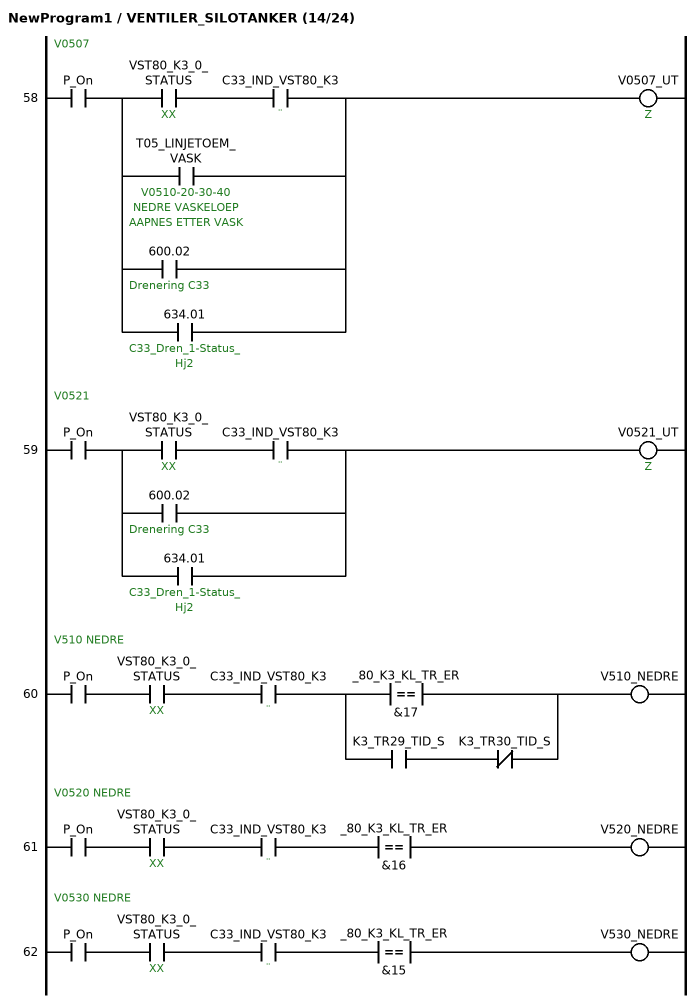
; [picture p864: NewProgram1 / VENTILER_SILOTANKER, rungs 58-62]
; rung 58: V0507
LD P_On
LD VST80_K3_0_STATUS  ; XX
AND C33_IND_VST80_K3  ; ¨
OR T05_LINJETOEM_VASK  ; V0510-20-30-40 NEDRE VASKELOEP AAPNES ETTER VASK
OR 600.02  ; Drenering C33
OR 634.01  ; C33_Dren_1-Status_Hj2
ANDLD
OUT V0507_UT  ; Z
; rung 59: V0521
LD P_On
LD VST80_K3_0_STATUS  ; XX
AND C33_IND_VST80_K3  ; ¨
OR 600.02  ; Drenering C33
OR 634.01  ; C33_Dren_1-Status_Hj2
ANDLD
OUT V0521_UT  ; Z
; rung 60: V510 NEDRE
LD P_On
AND VST80_K3_0_STATUS  ; XX
AND C33_IND_VST80_K3  ; ¨
LD=(300) _80_K3_KL_TR_ER &17
LD K3_TR29_TID_S
ANDNOT K3_TR30_TID_S
ORLD
ANDLD
OUT V510_NEDRE
; rung 61: V0520 NEDRE
LD P_On
AND VST80_K3_0_STATUS  ; XX
AND C33_IND_VST80_K3  ; ¨
AND=(300) _80_K3_KL_TR_ER &16
OUT V520_NEDRE
; rung 62: V0530 NEDRE
LD P_On
AND VST80_K3_0_STATUS  ; XX
AND C33_IND_VST80_K3  ; ¨
AND=(300) _80_K3_KL_TR_ER &15
OUT V530_NEDRE

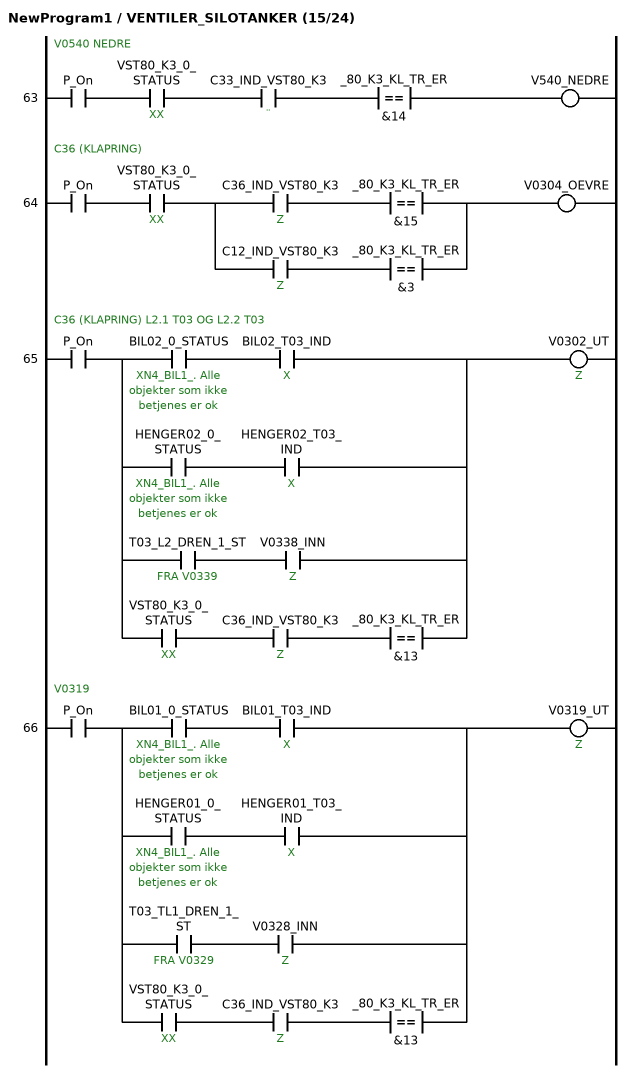
; rung 63: V0540 NEDRE
LD P_On
AND VST80_K3_0_STATUS  ; XX
AND C33_IND_VST80_K3  ; ¨
AND=(300) _80_K3_KL_TR_ER &14
OUT V540_NEDRE
; rung 64: C36 (KLAPRING)
LD P_On
AND VST80_K3_0_STATUS  ; XX
LD C36_IND_VST80_K3  ; Z
AND=(300) _80_K3_KL_TR_ER &15
LD C12_IND_VST80_K3  ; Z
AND=(300) _80_K3_KL_TR_ER &3
ORLD
ANDLD
OUT V0304_OEVRE
; rung 65: C36 (KLAPRING) L2.1 T03 OG L2.2 T03
LD P_On
LD BIL02_0_STATUS  ; XN4_BIL1_. Alle objekter som ikke betjenes er ok
AND BIL02_T03_IND  ; X
LD HENGER02_0_STATUS  ; XN4_BIL1_. Alle objekter som ikke betjenes er ok
AND HENGER02_T03_IND  ; X
ORLD
LD T03_L2_DREN_1_ST  ; FRA V0339
AND V0338_INN  ; Z
ORLD
LD VST80_K3_0_STATUS  ; XX
AND C36_IND_VST80_K3  ; Z
AND=(300) _80_K3_KL_TR_ER &13
ORLD
ANDLD
OUT V0302_UT  ; Z
; rung 66: V0319
LD P_On
LD BIL01_0_STATUS  ; XN4_BIL1_. Alle objekter som ikke betjenes er ok
AND BIL01_T03_IND  ; X
LD HENGER01_0_STATUS  ; XN4_BIL1_. Alle objekter som ikke betjenes er ok
AND HENGER01_T03_IND  ; X
ORLD
LD T03_TL1_DREN_1_ST  ; FRA V0329
AND V0328_INN  ; Z
ORLD
LD VST80_K3_0_STATUS  ; XX
AND C36_IND_VST80_K3  ; Z
AND=(300) _80_K3_KL_TR_ER &13
ORLD
ANDLD
OUT V0319_UT  ; Z

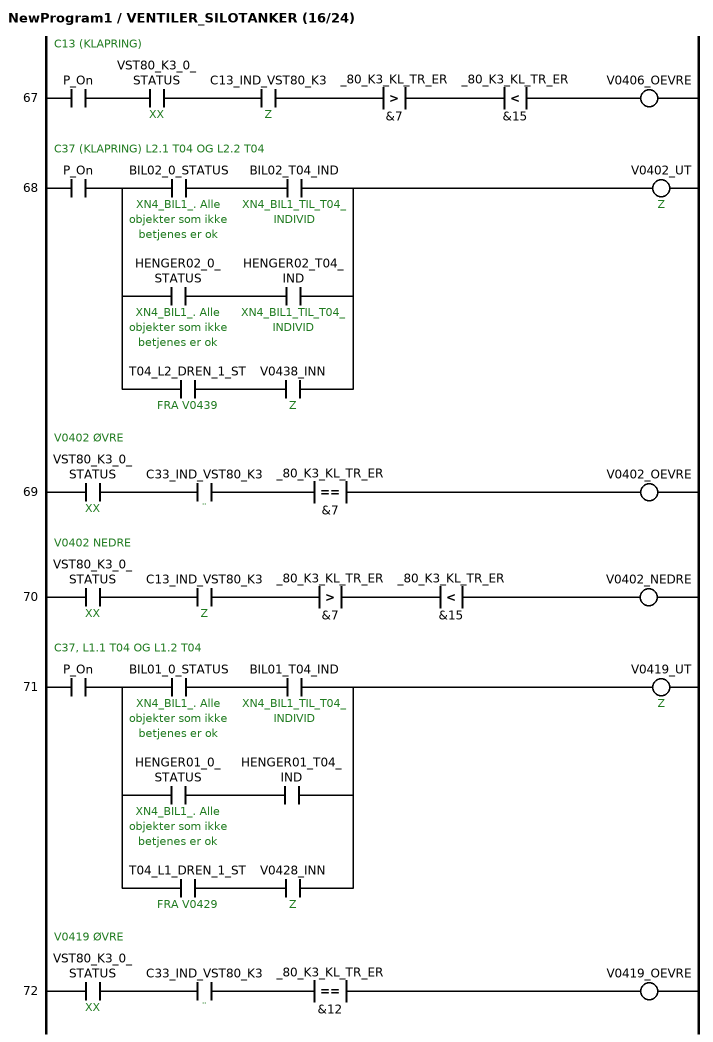
; rung 67: C13 (KLAPRING)
LD P_On
AND VST80_K3_0_STATUS  ; XX
AND C13_IND_VST80_K3  ; Z
AND>(320) _80_K3_KL_TR_ER &7
AND<(310) _80_K3_KL_TR_ER &15
OUT V0406_OEVRE
; rung 68: C37 (KLAPRING) L2.1 T04 OG L2.2 T04
LD P_On
LD BIL02_0_STATUS  ; XN4_BIL1_. Alle objekter som ikke betjenes er ok
AND BIL02_T04_IND  ; XN4_BIL1_TIL_T04_INDIVID
LD HENGER02_0_STATUS  ; XN4_BIL1_. Alle objekter som ikke betjenes er ok
AND HENGER02_T04_IND  ; XN4_BIL1_TIL_T04_INDIVID
ORLD
LD T04_L2_DREN_1_ST  ; FRA V0439
AND V0438_INN  ; Z
ORLD
ANDLD
OUT V0402_UT  ; Z
; rung 69: V0402 ØVRE
LD VST80_K3_0_STATUS  ; XX
AND C33_IND_VST80_K3  ; ¨
AND=(300) _80_K3_KL_TR_ER &7
OUT V0402_OEVRE
; rung 70: V0402 NEDRE
LD VST80_K3_0_STATUS  ; XX
AND C13_IND_VST80_K3  ; Z
AND>(320) _80_K3_KL_TR_ER &7
AND<(310) _80_K3_KL_TR_ER &15
OUT V0402_NEDRE
; rung 71: C37, L1.1 T04 OG L1.2 T04
LD P_On
LD BIL01_0_STATUS  ; XN4_BIL1_. Alle objekter som ikke betjenes er ok
AND BIL01_T04_IND  ; XN4_BIL1_TIL_T04_INDIVID
LD HENGER01_0_STATUS  ; XN4_BIL1_. Alle objekter som ikke betjenes er ok
AND HENGER01_T04_IND
ORLD
LD T04_L1_DREN_1_ST  ; FRA V0429
AND V0428_INN  ; Z
ORLD
ANDLD
OUT V0419_UT  ; Z
; rung 72: V0419 ØVRE
LD VST80_K3_0_STATUS  ; XX
AND C33_IND_VST80_K3  ; ¨
AND=(300) _80_K3_KL_TR_ER &12
OUT V0419_OEVRE

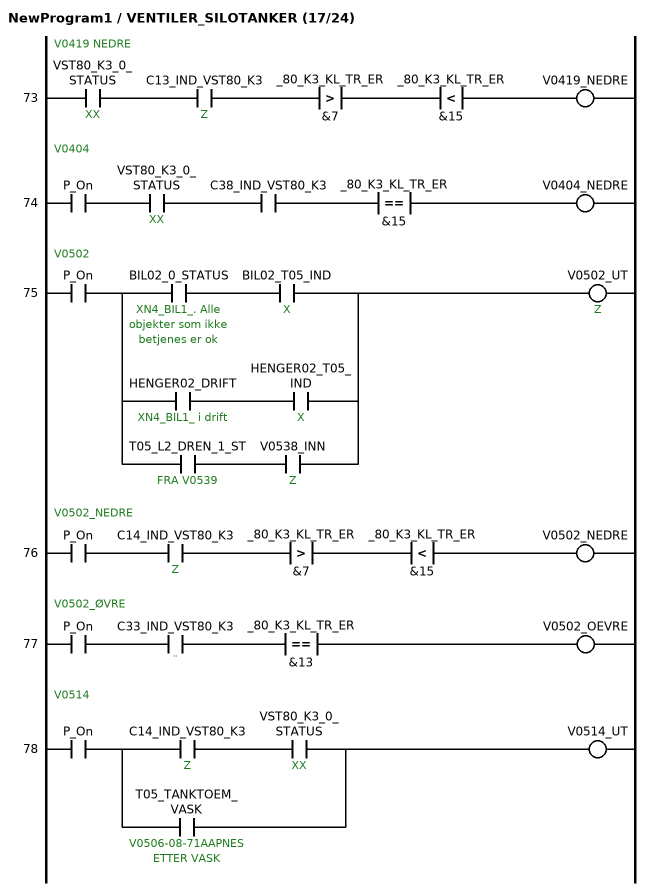
; rung 73: V0419 NEDRE
LD VST80_K3_0_STATUS  ; XX
AND C13_IND_VST80_K3  ; Z
AND>(320) _80_K3_KL_TR_ER &7
AND<(310) _80_K3_KL_TR_ER &15
OUT V0419_NEDRE
; rung 74: V0404
LD P_On
AND VST80_K3_0_STATUS  ; XX
AND C38_IND_VST80_K3
AND=(300) _80_K3_KL_TR_ER &15
OUT V0404_NEDRE
; rung 75: V0502
LD P_On
LD BIL02_0_STATUS  ; XN4_BIL1_. Alle objekter som ikke betjenes er ok
AND BIL02_T05_IND  ; X
LD HENGER02_DRIFT  ; XN4_BIL1_ i drift
AND HENGER02_T05_IND  ; X
ORLD
LD T05_L2_DREN_1_ST  ; FRA V0539
AND V0538_INN  ; Z
ORLD
ANDLD
OUT V0502_UT  ; Z
; rung 76: V0502_NEDRE
LD P_On
AND C14_IND_VST80_K3  ; Z
AND>(320) _80_K3_KL_TR_ER &7
AND<(310) _80_K3_KL_TR_ER &15
OUT V0502_NEDRE
; rung 77: V0502_ØVRE
LD P_On
AND C33_IND_VST80_K3  ; ¨
AND=(300) _80_K3_KL_TR_ER &13
OUT V0502_OEVRE
; rung 78: V0514
LD P_On
LD C14_IND_VST80_K3  ; Z
AND VST80_K3_0_STATUS  ; XX
OR T05_TANKTOEM_VASK  ; V0506-08-71AAPNES ETTER VASK
ANDLD
OUT V0514_UT

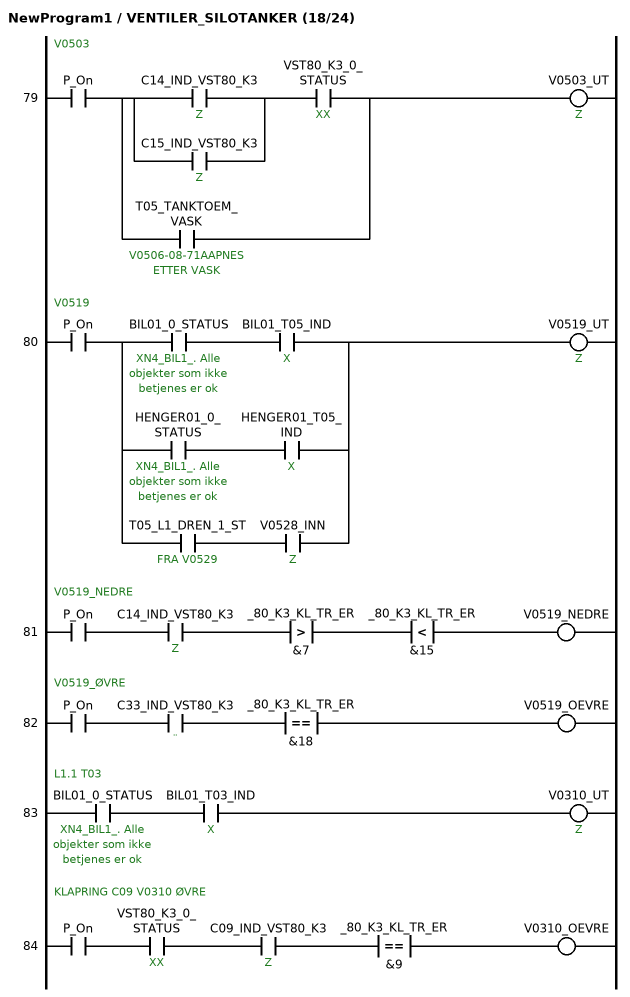
; rung 79: V0503
LD P_On
LD C14_IND_VST80_K3  ; Z
OR C15_IND_VST80_K3  ; Z
AND VST80_K3_0_STATUS  ; XX
OR T05_TANKTOEM_VASK  ; V0506-08-71AAPNES ETTER VASK
ANDLD
OUT V0503_UT  ; Z
; rung 80: V0519
LD P_On
LD BIL01_0_STATUS  ; XN4_BIL1_. Alle objekter som ikke betjenes er ok
AND BIL01_T05_IND  ; X
LD HENGER01_0_STATUS  ; XN4_BIL1_. Alle objekter som ikke betjenes er ok
AND HENGER01_T05_IND  ; X
ORLD
LD T05_L1_DREN_1_ST  ; FRA V0529
AND V0528_INN  ; Z
ORLD
ANDLD
OUT V0519_UT  ; Z
; rung 81: V0519_NEDRE
LD P_On
AND C14_IND_VST80_K3  ; Z
AND>(320) _80_K3_KL_TR_ER &7
AND<(310) _80_K3_KL_TR_ER &15
OUT V0519_NEDRE
; rung 82: V0519_ØVRE
LD P_On
AND C33_IND_VST80_K3  ; ¨
AND=(300) _80_K3_KL_TR_ER &18
OUT V0519_OEVRE
; rung 83: L1.1 T03
LD BIL01_0_STATUS  ; XN4_BIL1_. Alle objekter som ikke betjenes er ok
AND BIL01_T03_IND  ; X
OUT V0310_UT  ; Z
; rung 84: KLAPRING C09 V0310 ØVRE
LD P_On
AND VST80_K3_0_STATUS  ; XX
AND C09_IND_VST80_K3  ; Z
AND=(300) _80_K3_KL_TR_ER &9
OUT V0310_OEVRE

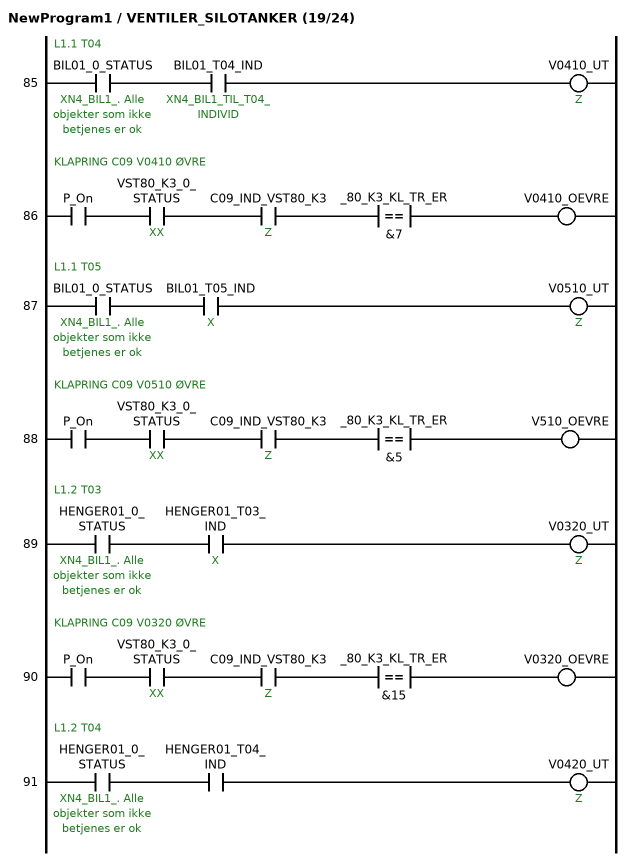
; rung 85: L1.1 T04
LD BIL01_0_STATUS  ; XN4_BIL1_. Alle objekter som ikke betjenes er ok
AND BIL01_T04_IND  ; XN4_BIL1_TIL_T04_INDIVID
OUT V0410_UT  ; Z
; rung 86: KLAPRING C09 V0410 ØVRE
LD P_On
AND VST80_K3_0_STATUS  ; XX
AND C09_IND_VST80_K3  ; Z
AND=(300) _80_K3_KL_TR_ER &7
OUT V0410_OEVRE
; rung 87: L1.1 T05
LD BIL01_0_STATUS  ; XN4_BIL1_. Alle objekter som ikke betjenes er ok
AND BIL01_T05_IND  ; X
OUT V0510_UT  ; Z
; rung 88: KLAPRING C09 V0510 ØVRE
LD P_On
AND VST80_K3_0_STATUS  ; XX
AND C09_IND_VST80_K3  ; Z
AND=(300) _80_K3_KL_TR_ER &5
OUT V510_OEVRE
; rung 89: L1.2 T03
LD HENGER01_0_STATUS  ; XN4_BIL1_. Alle objekter som ikke betjenes er ok
AND HENGER01_T03_IND  ; X
OUT V0320_UT  ; Z
; rung 90: KLAPRING C09 V0320 ØVRE
LD P_On
AND VST80_K3_0_STATUS  ; XX
AND C09_IND_VST80_K3  ; Z
AND=(300) _80_K3_KL_TR_ER &15
OUT V0320_OEVRE
; rung 91: L1.2 T04
LD HENGER01_0_STATUS  ; XN4_BIL1_. Alle objekter som ikke betjenes er ok
AND HENGER01_T04_IND
OUT V0420_UT  ; Z

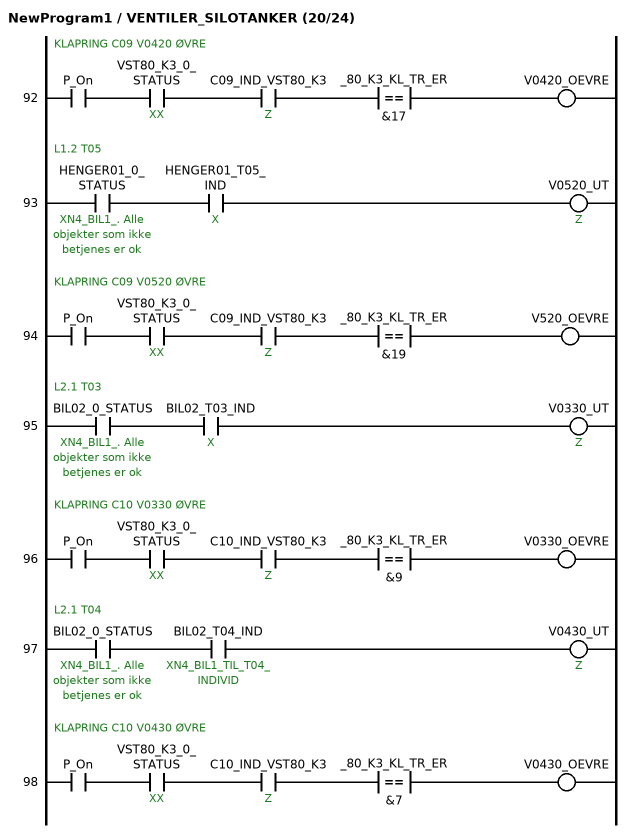
; rung 92: KLAPRING C09 V0420 ØVRE
LD P_On
AND VST80_K3_0_STATUS  ; XX
AND C09_IND_VST80_K3  ; Z
AND=(300) _80_K3_KL_TR_ER &17
OUT V0420_OEVRE
; rung 93: L1.2 T05
LD HENGER01_0_STATUS  ; XN4_BIL1_. Alle objekter som ikke betjenes er ok
AND HENGER01_T05_IND  ; X
OUT V0520_UT  ; Z
; rung 94: KLAPRING C09 V0520 ØVRE
LD P_On
AND VST80_K3_0_STATUS  ; XX
AND C09_IND_VST80_K3  ; Z
AND=(300) _80_K3_KL_TR_ER &19
OUT V520_OEVRE
; rung 95: L2.1 T03
LD BIL02_0_STATUS  ; XN4_BIL1_. Alle objekter som ikke betjenes er ok
AND BIL02_T03_IND  ; X
OUT V0330_UT  ; Z
; rung 96: KLAPRING C10 V0330 ØVRE
LD P_On
AND VST80_K3_0_STATUS  ; XX
AND C10_IND_VST80_K3  ; Z
AND=(300) _80_K3_KL_TR_ER &9
OUT V0330_OEVRE
; rung 97: L2.1 T04
LD BIL02_0_STATUS  ; XN4_BIL1_. Alle objekter som ikke betjenes er ok
AND BIL02_T04_IND  ; XN4_BIL1_TIL_T04_INDIVID
OUT V0430_UT  ; Z
; rung 98: KLAPRING C10 V0430 ØVRE
LD P_On
AND VST80_K3_0_STATUS  ; XX
AND C10_IND_VST80_K3  ; Z
AND=(300) _80_K3_KL_TR_ER &7
OUT V0430_OEVRE

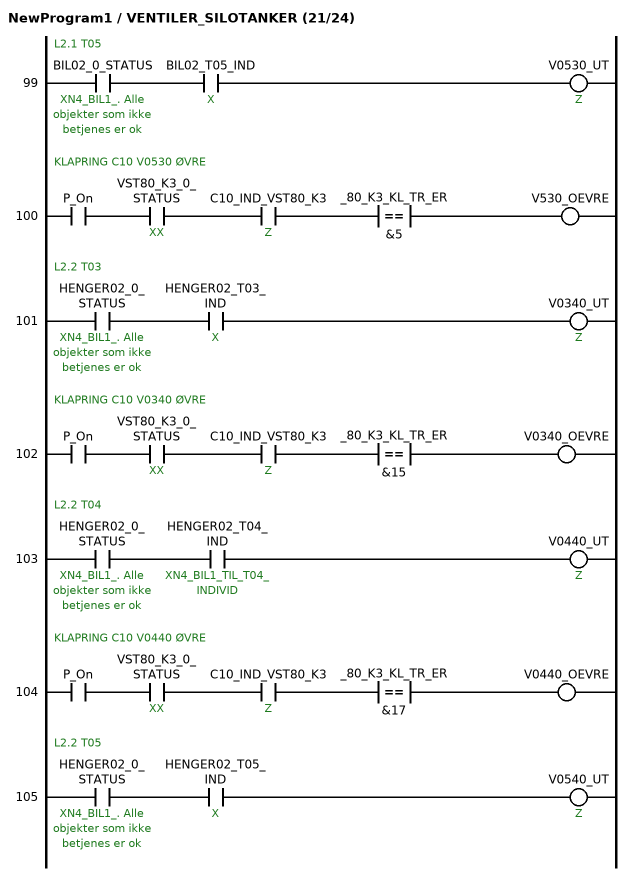
; rung 99: L2.1 T05
LD BIL02_0_STATUS  ; XN4_BIL1_. Alle objekter som ikke betjenes er ok
AND BIL02_T05_IND  ; X
OUT V0530_UT  ; Z
; rung 100: KLAPRING C10 V0530 ØVRE
LD P_On
AND VST80_K3_0_STATUS  ; XX
AND C10_IND_VST80_K3  ; Z
AND=(300) _80_K3_KL_TR_ER &5
OUT V530_OEVRE
; rung 101: L2.2 T03
LD HENGER02_0_STATUS  ; XN4_BIL1_. Alle objekter som ikke betjenes er ok
AND HENGER02_T03_IND  ; X
OUT V0340_UT  ; Z
; rung 102: KLAPRING C10 V0340 ØVRE
LD P_On
AND VST80_K3_0_STATUS  ; XX
AND C10_IND_VST80_K3  ; Z
AND=(300) _80_K3_KL_TR_ER &15
OUT V0340_OEVRE
; rung 103: L2.2 T04
LD HENGER02_0_STATUS  ; XN4_BIL1_. Alle objekter som ikke betjenes er ok
AND HENGER02_T04_IND  ; XN4_BIL1_TIL_T04_INDIVID
OUT V0440_UT  ; Z
; rung 104: KLAPRING C10 V0440 ØVRE
LD P_On
AND VST80_K3_0_STATUS  ; XX
AND C10_IND_VST80_K3  ; Z
AND=(300) _80_K3_KL_TR_ER &17
OUT V0440_OEVRE
; rung 105: L2.2 T05
LD HENGER02_0_STATUS  ; XN4_BIL1_. Alle objekter som ikke betjenes er ok
AND HENGER02_T05_IND  ; X
OUT V0540_UT  ; Z

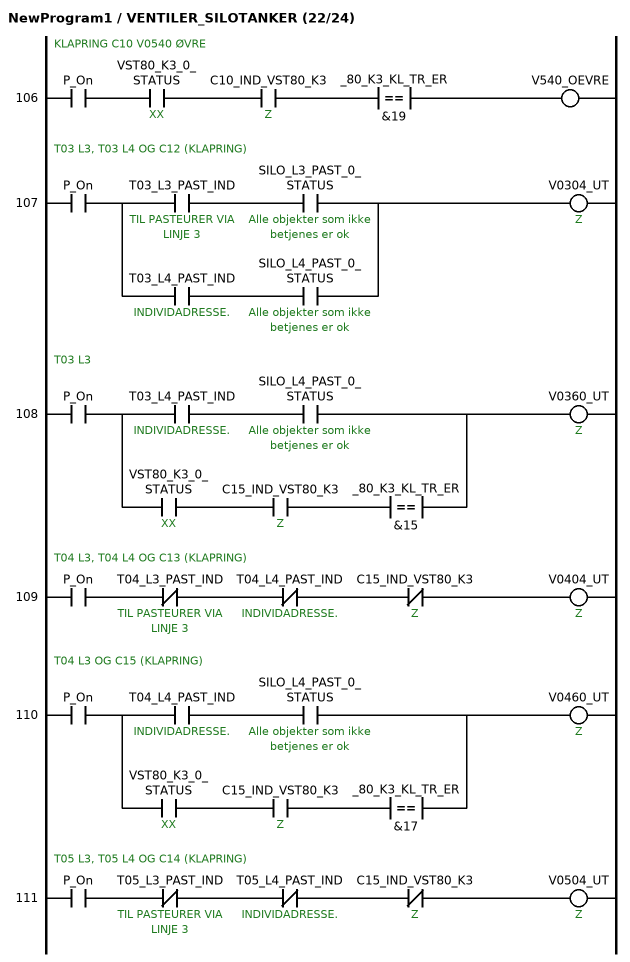
; rung 106: KLAPRING C10 V0540 ØVRE
LD P_On
AND VST80_K3_0_STATUS  ; XX
AND C10_IND_VST80_K3  ; Z
AND=(300) _80_K3_KL_TR_ER &19
OUT V540_OEVRE
; rung 107: T03 L3, T03 L4 OG C12 (KLAPRING)
LD P_On
LD T03_L3_PAST_IND  ; TIL PASTEURER VIA LINJE 3
AND SILO_L3_PAST_0_STATUS  ; Alle objekter som ikke betjenes er ok
LD T03_L4_PAST_IND  ; INDIVIDADRESSE.
AND SILO_L4_PAST_0_STATUS  ; Alle objekter som ikke betjenes er ok
ORLD
ANDLD
OUT V0304_UT  ; Z
; rung 108: T03 L3
LD P_On
LD T03_L4_PAST_IND  ; INDIVIDADRESSE.
AND SILO_L4_PAST_0_STATUS  ; Alle objekter som ikke betjenes er ok
LD VST80_K3_0_STATUS  ; XX
AND C15_IND_VST80_K3  ; Z
AND=(300) _80_K3_KL_TR_ER &15
ORLD
ANDLD
OUT V0360_UT  ; Z
; rung 109: T04 L3, T04 L4 OG C13 (KLAPRING)
LD P_On
ANDNOT T04_L3_PAST_IND  ; TIL PASTEURER VIA LINJE 3
ANDNOT T04_L4_PAST_IND  ; INDIVIDADRESSE.
ANDNOT C15_IND_VST80_K3  ; Z
OUT V0404_UT  ; Z
; rung 110: T04 L3 OG C15 (KLAPRING)
LD P_On
LD T04_L4_PAST_IND  ; INDIVIDADRESSE.
AND SILO_L4_PAST_0_STATUS  ; Alle objekter som ikke betjenes er ok
LD VST80_K3_0_STATUS  ; XX
AND C15_IND_VST80_K3  ; Z
AND=(300) _80_K3_KL_TR_ER &17
ORLD
ANDLD
OUT V0460_UT  ; Z
; rung 111: T05 L3, T05 L4 OG C14 (KLAPRING)
LD P_On
ANDNOT T05_L3_PAST_IND  ; TIL PASTEURER VIA LINJE 3
ANDNOT T05_L4_PAST_IND  ; INDIVIDADRESSE.
ANDNOT C15_IND_VST80_K3  ; Z
OUT V0504_UT  ; Z

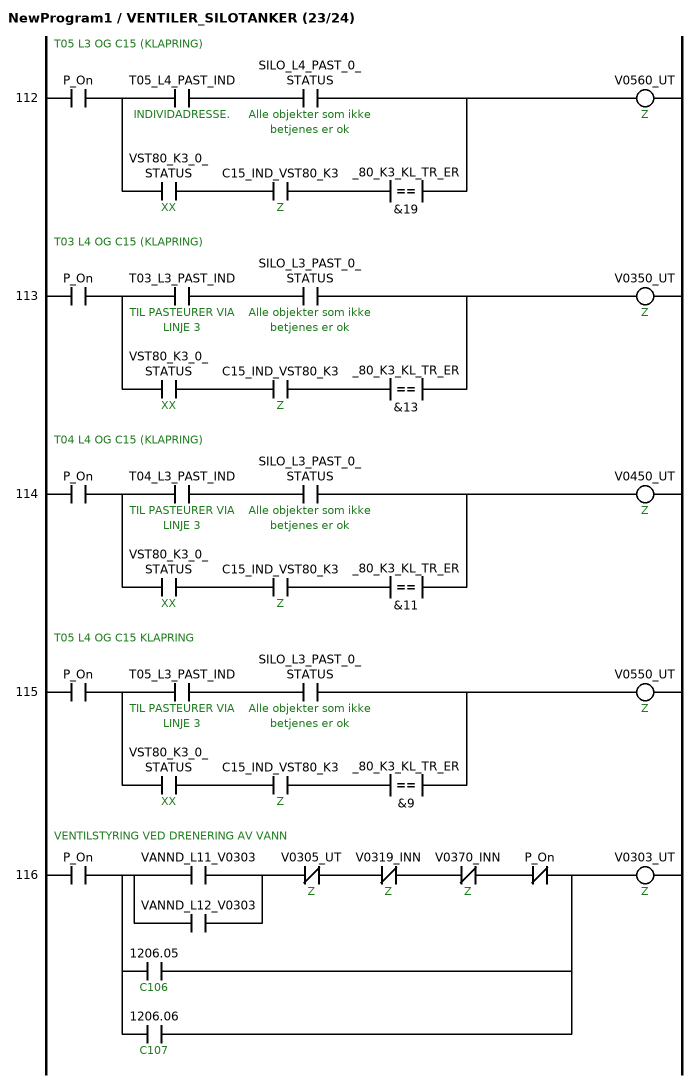
; rung 112: T05 L3 OG C15 (KLAPRING)
LD P_On
LD T05_L4_PAST_IND  ; INDIVIDADRESSE.
AND SILO_L4_PAST_0_STATUS  ; Alle objekter som ikke betjenes er ok
LD VST80_K3_0_STATUS  ; XX
AND C15_IND_VST80_K3  ; Z
AND=(300) _80_K3_KL_TR_ER &19
ORLD
ANDLD
OUT V0560_UT  ; Z
; rung 113: T03 L4 OG C15 (KLAPRING)
LD P_On
LD T03_L3_PAST_IND  ; TIL PASTEURER VIA LINJE 3
AND SILO_L3_PAST_0_STATUS  ; Alle objekter som ikke betjenes er ok
LD VST80_K3_0_STATUS  ; XX
AND C15_IND_VST80_K3  ; Z
AND=(300) _80_K3_KL_TR_ER &13
ORLD
ANDLD
OUT V0350_UT  ; Z
; rung 114: T04 L4 OG C15 (KLAPRING)
LD P_On
LD T04_L3_PAST_IND  ; TIL PASTEURER VIA LINJE 3
AND SILO_L3_PAST_0_STATUS  ; Alle objekter som ikke betjenes er ok
LD VST80_K3_0_STATUS  ; XX
AND C15_IND_VST80_K3  ; Z
AND=(300) _80_K3_KL_TR_ER &11
ORLD
ANDLD
OUT V0450_UT  ; Z
; rung 115: T05 L4 OG C15 KLAPRING
LD P_On
LD T05_L3_PAST_IND  ; TIL PASTEURER VIA LINJE 3
AND SILO_L3_PAST_0_STATUS  ; Alle objekter som ikke betjenes er ok
LD VST80_K3_0_STATUS  ; XX
AND C15_IND_VST80_K3  ; Z
AND=(300) _80_K3_KL_TR_ER &9
ORLD
ANDLD
OUT V0550_UT  ; Z
; rung 116: VENTILSTYRING VED DRENERING AV VANN
LD P_On
LD VANND_L11_V0303
OR VANND_L12_V0303
ANDNOT V0305_UT  ; Z
ANDNOT V0319_INN  ; Z
ANDNOT V0370_INN  ; Z
ANDNOT P_On
OR 1206.05  ; C106
OR 1206.06  ; C107
ANDLD
OUT V0303_UT  ; Z

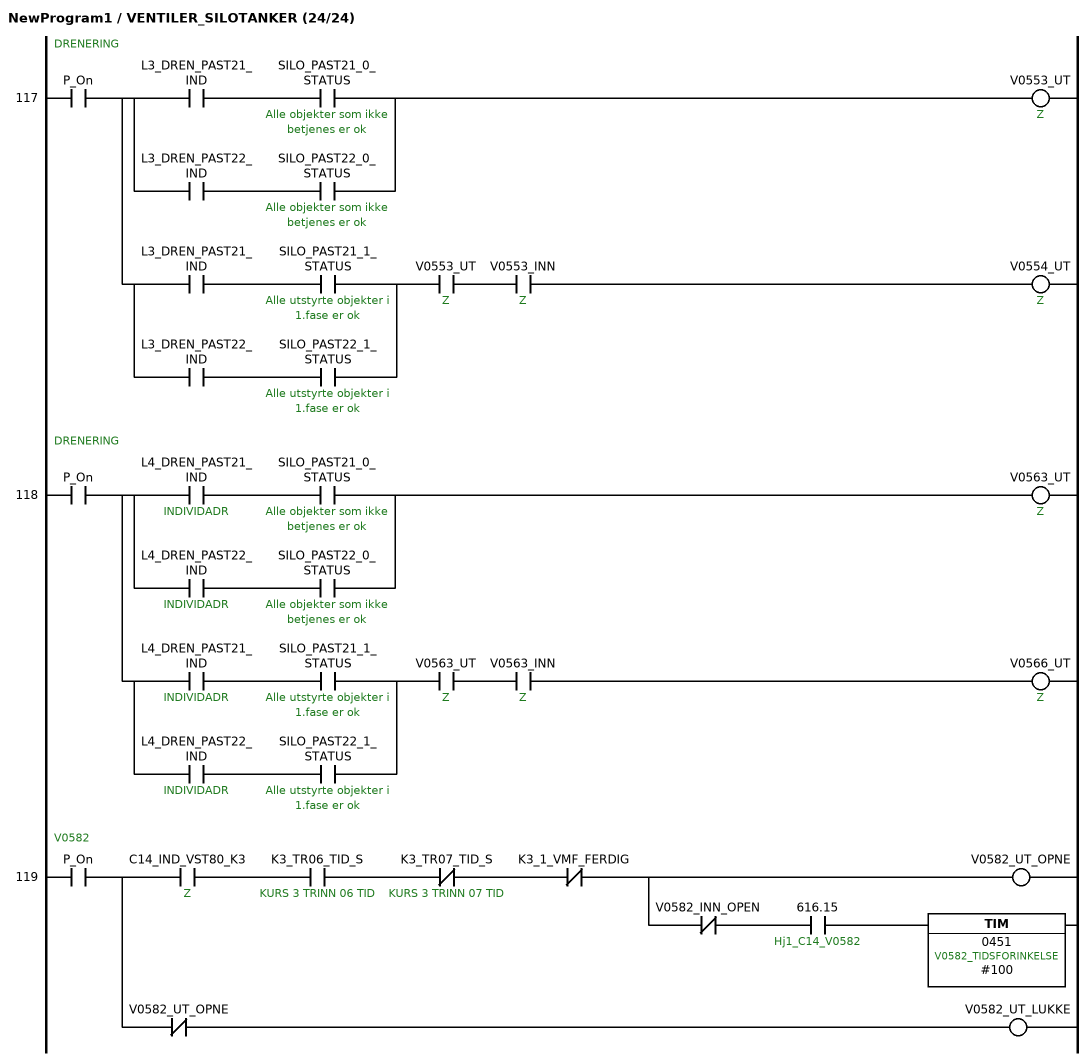
; rung 117: DRENERING
LD P_On
OUT TR0
LD L3_DREN_PAST21_IND
AND SILO_PAST21_0_STATUS  ; Alle objekter som ikke betjenes er ok
LD L3_DREN_PAST22_IND
AND SILO_PAST22_0_STATUS  ; Alle objekter som ikke betjenes er ok
ORLD
ANDLD
OUT V0553_UT  ; Z
LD TR0
LD L3_DREN_PAST21_IND
AND SILO_PAST21_1_STATUS  ; Alle utstyrte objekter i 1.fase er ok
LD L3_DREN_PAST22_IND
AND SILO_PAST22_1_STATUS  ; Alle utstyrte objekter i 1.fase er ok
ORLD
ANDLD
AND V0553_UT  ; Z
AND V0553_INN  ; Z
OUT V0554_UT  ; Z
; rung 118: DRENERING
LD P_On
OUT TR0
LD L4_DREN_PAST21_IND  ; INDIVIDADR
AND SILO_PAST21_0_STATUS  ; Alle objekter som ikke betjenes er ok
LD L4_DREN_PAST22_IND  ; INDIVIDADR
AND SILO_PAST22_0_STATUS  ; Alle objekter som ikke betjenes er ok
ORLD
ANDLD
OUT V0563_UT  ; Z
LD TR0
LD L4_DREN_PAST21_IND  ; INDIVIDADR
AND SILO_PAST21_1_STATUS  ; Alle utstyrte objekter i 1.fase er ok
LD L4_DREN_PAST22_IND  ; INDIVIDADR
AND SILO_PAST22_1_STATUS  ; Alle utstyrte objekter i 1.fase er ok
ORLD
ANDLD
AND V0563_UT  ; Z
AND V0563_INN  ; Z
OUT V0566_UT  ; Z
; rung 119: V0582
LD P_On
OUT TR0
AND C14_IND_VST80_K3  ; Z
AND K3_TR06_TID_S  ; KURS 3 TRINN 06 TID
ANDNOT K3_TR07_TID_S  ; KURS 3 TRINN 07 TID
ANDNOT K3_1_VMF_FERDIG
OUT V0582_UT_OPNE
ANDNOT V0582_INN_OPEN
AND 616.15  ; Hj1_C14_V0582
TIM 0451 #100  ; V0582_TIDSFORINKELSE
LD TR0
ANDNOT V0582_UT_OPNE
OUT V0582_UT_LUKKE
; rung 120: Ingen_kommentar_funnet

### Section VENTILER_PROD_MOTTAK

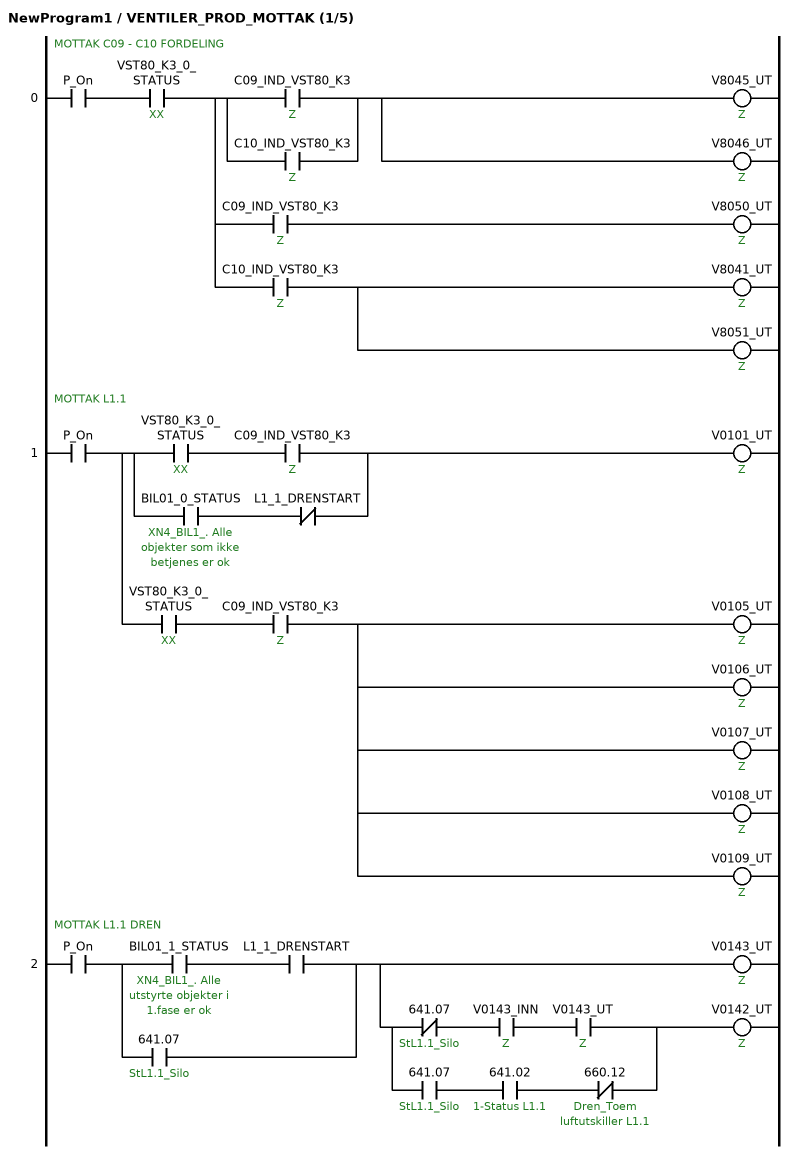
; rung 0: MOTTAK C09 - C10 FORDELING
LD P_On
AND VST80_K3_0_STATUS  ; XX
OUT TR0
LD C09_IND_VST80_K3  ; Z
OR C10_IND_VST80_K3  ; Z
ANDLD
OUT V8045_UT  ; Z
OUT V8046_UT  ; Z
LD TR0
AND C09_IND_VST80_K3  ; Z
OUT V8050_UT  ; Z
LD TR0
AND C10_IND_VST80_K3  ; Z
OUT V8041_UT  ; Z
OUT V8051_UT  ; Z
; rung 1: MOTTAK L1.1
LD P_On
OUT TR0
LD VST80_K3_0_STATUS  ; XX
AND C09_IND_VST80_K3  ; Z
LD BIL01_0_STATUS  ; XN4_BIL1_. Alle objekter som ikke betjenes er ok
ANDNOT L1_1_DRENSTART
ORLD
ANDLD
OUT V0101_UT  ; Z
LD TR0
AND VST80_K3_0_STATUS  ; XX
AND C09_IND_VST80_K3  ; Z
OUT V0105_UT  ; Z
OUT V0106_UT  ; Z
OUT V0107_UT  ; Z
OUT V0108_UT  ; Z
OUT V0109_UT  ; Z
; rung 2: MOTTAK L1.1 DREN
LD P_On
LD BIL01_1_STATUS  ; XN4_BIL1_. Alle utstyrte objekter i 1.fase er ok
AND L1_1_DRENSTART
OR 641.07  ; StL1.1_Silo
ANDLD
OUT V0143_UT  ; Z
LDNOT 641.07  ; StL1.1_Silo
AND V0143_INN  ; Z
AND V0143_UT  ; Z
LD 641.07  ; StL1.1_Silo
AND 641.02  ; 1-Status L1.1
ANDNOT 660.12  ; Dren_Toem luftutskiller L1.1
ORLD
ANDLD
OUT V0142_UT  ; Z

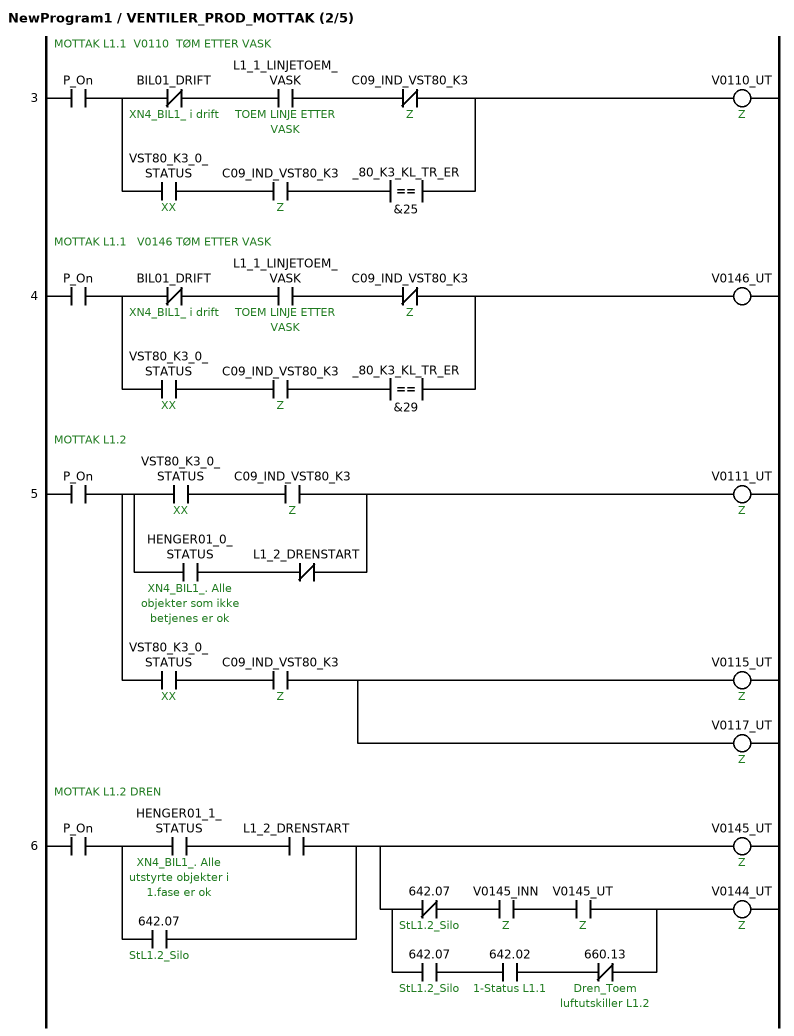
; rung 3: MOTTAK L1.1  V0110  TØM ETTER VASK
LD P_On
LDNOT BIL01_DRIFT  ; XN4_BIL1_ i drift
AND L1_1_LINJETOEM_VASK  ; TOEM LINJE ETTER VASK
ANDNOT C09_IND_VST80_K3  ; Z
LD VST80_K3_0_STATUS  ; XX
AND C09_IND_VST80_K3  ; Z
AND=(300) _80_K3_KL_TR_ER &25
ORLD
ANDLD
OUT V0110_UT  ; Z
; rung 4: MOTTAK L1.1   V0146 TØM ETTER VASK
LD P_On
LDNOT BIL01_DRIFT  ; XN4_BIL1_ i drift
AND L1_1_LINJETOEM_VASK  ; TOEM LINJE ETTER VASK
ANDNOT C09_IND_VST80_K3  ; Z
LD VST80_K3_0_STATUS  ; XX
AND C09_IND_VST80_K3  ; Z
AND=(300) _80_K3_KL_TR_ER &29
ORLD
ANDLD
OUT V0146_UT
; rung 5: MOTTAK L1.2
LD P_On
OUT TR0
LD VST80_K3_0_STATUS  ; XX
AND C09_IND_VST80_K3  ; Z
LD HENGER01_0_STATUS  ; XN4_BIL1_. Alle objekter som ikke betjenes er ok
ANDNOT L1_2_DRENSTART
ORLD
ANDLD
OUT V0111_UT  ; Z
LD TR0
AND VST80_K3_0_STATUS  ; XX
AND C09_IND_VST80_K3  ; Z
OUT V0115_UT  ; Z
OUT V0117_UT  ; Z
; rung 6: MOTTAK L1.2 DREN
LD P_On
LD HENGER01_1_STATUS  ; XN4_BIL1_. Alle utstyrte objekter i 1.fase er ok
AND L1_2_DRENSTART
OR 642.07  ; StL1.2_Silo
ANDLD
OUT V0145_UT  ; Z
LDNOT 642.07  ; StL1.2_Silo
AND V0145_INN  ; Z
AND V0145_UT  ; Z
LD 642.07  ; StL1.2_Silo
AND 642.02  ; 1-Status L1.1
ANDNOT 660.13  ; Dren_Toem luftutskiller L1.2
ORLD
ANDLD
OUT V0144_UT  ; Z

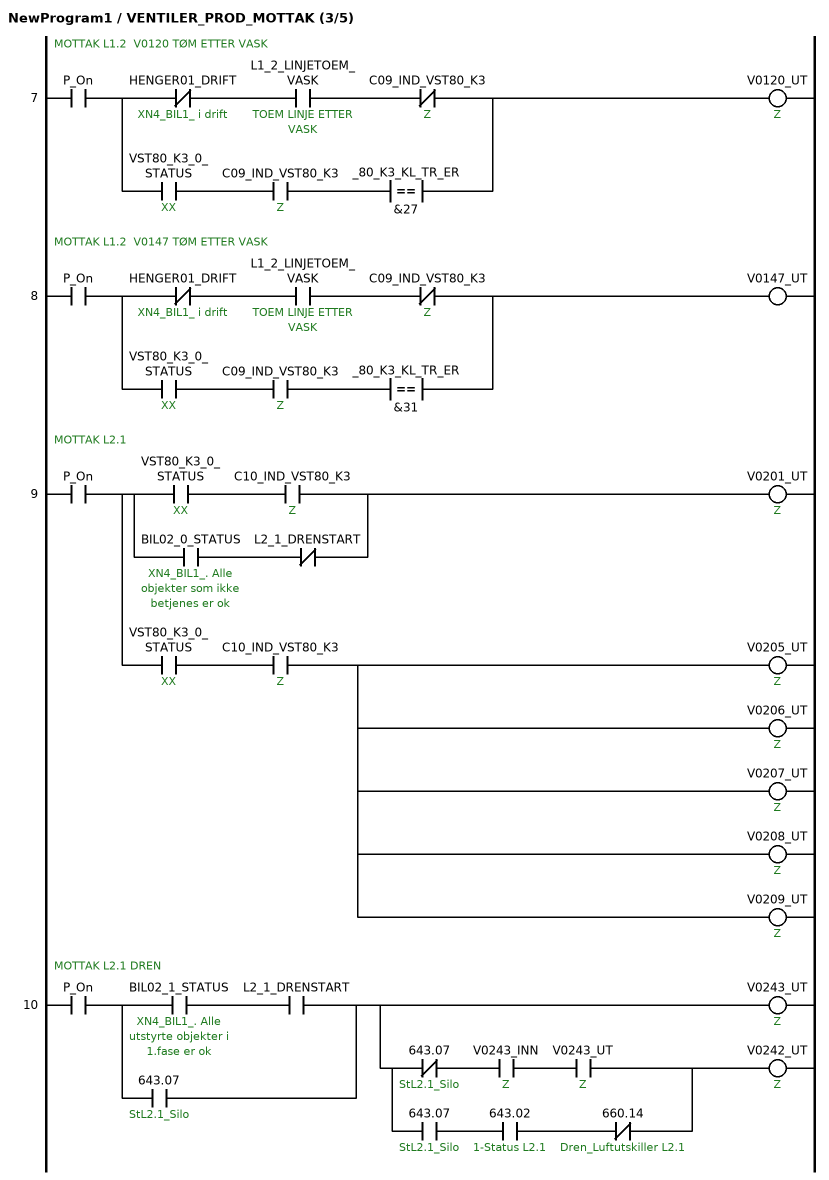
; rung 7: MOTTAK L1.2  V0120 TØM ETTER VASK
LD P_On
LDNOT HENGER01_DRIFT  ; XN4_BIL1_ i drift
AND L1_2_LINJETOEM_VASK  ; TOEM LINJE ETTER VASK
ANDNOT C09_IND_VST80_K3  ; Z
LD VST80_K3_0_STATUS  ; XX
AND C09_IND_VST80_K3  ; Z
AND=(300) _80_K3_KL_TR_ER &27
ORLD
ANDLD
OUT V0120_UT  ; Z
; rung 8: MOTTAK L1.2  V0147 TØM ETTER VASK
LD P_On
LDNOT HENGER01_DRIFT  ; XN4_BIL1_ i drift
AND L1_2_LINJETOEM_VASK  ; TOEM LINJE ETTER VASK
ANDNOT C09_IND_VST80_K3  ; Z
LD VST80_K3_0_STATUS  ; XX
AND C09_IND_VST80_K3  ; Z
AND=(300) _80_K3_KL_TR_ER &31
ORLD
ANDLD
OUT V0147_UT
; rung 9: MOTTAK L2.1
LD P_On
OUT TR0
LD VST80_K3_0_STATUS  ; XX
AND C10_IND_VST80_K3  ; Z
LD BIL02_0_STATUS  ; XN4_BIL1_. Alle objekter som ikke betjenes er ok
ANDNOT L2_1_DRENSTART
ORLD
ANDLD
OUT V0201_UT  ; Z
LD TR0
AND VST80_K3_0_STATUS  ; XX
AND C10_IND_VST80_K3  ; Z
OUT V0205_UT  ; Z
OUT V0206_UT  ; Z
OUT V0207_UT  ; Z
OUT V0208_UT  ; Z
OUT V0209_UT  ; Z
; rung 10: MOTTAK L2.1 DREN
LD P_On
LD BIL02_1_STATUS  ; XN4_BIL1_. Alle utstyrte objekter i 1.fase er ok
AND L2_1_DRENSTART
OR 643.07  ; StL2.1_Silo
ANDLD
OUT V0243_UT  ; Z
LDNOT 643.07  ; StL2.1_Silo
AND V0243_INN  ; Z
AND V0243_UT  ; Z
LD 643.07  ; StL2.1_Silo
AND 643.02  ; 1-Status L2.1
ANDNOT 660.14  ; Dren_Luftutskiller L2.1
ORLD
ANDLD
OUT V0242_UT  ; Z

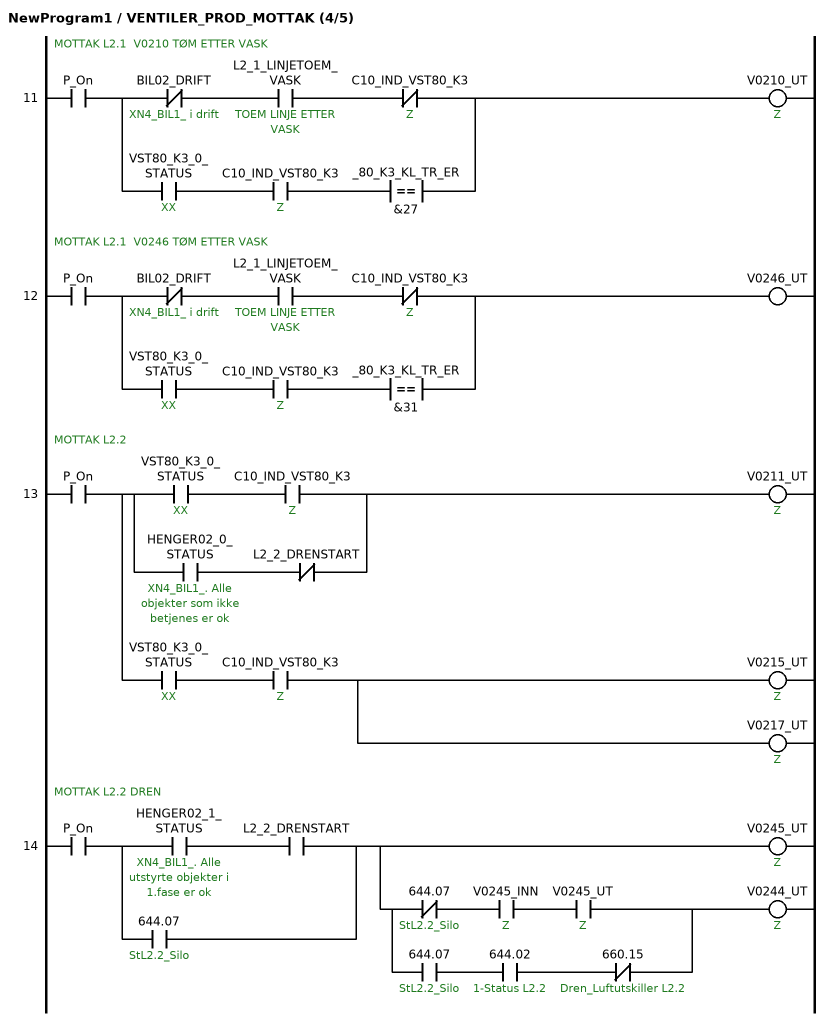
; rung 11: MOTTAK L2.1  V0210 TØM ETTER VASK
LD P_On
LDNOT BIL02_DRIFT  ; XN4_BIL1_ i drift
AND L2_1_LINJETOEM_VASK  ; TOEM LINJE ETTER VASK
ANDNOT C10_IND_VST80_K3  ; Z
LD VST80_K3_0_STATUS  ; XX
AND C10_IND_VST80_K3  ; Z
AND=(300) _80_K3_KL_TR_ER &27
ORLD
ANDLD
OUT V0210_UT  ; Z
; rung 12: MOTTAK L2.1  V0246 TØM ETTER VASK
LD P_On
LDNOT BIL02_DRIFT  ; XN4_BIL1_ i drift
AND L2_1_LINJETOEM_VASK  ; TOEM LINJE ETTER VASK
ANDNOT C10_IND_VST80_K3  ; Z
LD VST80_K3_0_STATUS  ; XX
AND C10_IND_VST80_K3  ; Z
AND=(300) _80_K3_KL_TR_ER &31
ORLD
ANDLD
OUT V0246_UT
; rung 13: MOTTAK L2.2
LD P_On
OUT TR0
LD VST80_K3_0_STATUS  ; XX
AND C10_IND_VST80_K3  ; Z
LD HENGER02_0_STATUS  ; XN4_BIL1_. Alle objekter som ikke betjenes er ok
ANDNOT L2_2_DRENSTART
ORLD
ANDLD
OUT V0211_UT  ; Z
LD TR0
AND VST80_K3_0_STATUS  ; XX
AND C10_IND_VST80_K3  ; Z
OUT V0215_UT  ; Z
OUT V0217_UT  ; Z
; rung 14: MOTTAK L2.2 DREN
LD P_On
LD HENGER02_1_STATUS  ; XN4_BIL1_. Alle utstyrte objekter i 1.fase er ok
AND L2_2_DRENSTART
OR 644.07  ; StL2.2_Silo
ANDLD
OUT V0245_UT  ; Z
LDNOT 644.07  ; StL2.2_Silo
AND V0245_INN  ; Z
AND V0245_UT  ; Z
LD 644.07  ; StL2.2_Silo
AND 644.02  ; 1-Status L2.2
ANDNOT 660.15  ; Dren_Luftutskiller L2.2
ORLD
ANDLD
OUT V0244_UT  ; Z

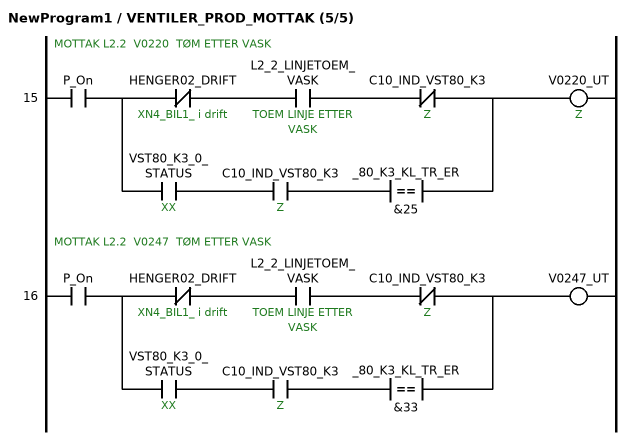
; rung 15: MOTTAK L2.2  V0220  TØM ETTER VASK
LD P_On
LDNOT HENGER02_DRIFT  ; XN4_BIL1_ i drift
AND L2_2_LINJETOEM_VASK  ; TOEM LINJE ETTER VASK
ANDNOT C10_IND_VST80_K3  ; Z
LD VST80_K3_0_STATUS  ; XX
AND C10_IND_VST80_K3  ; Z
AND=(300) _80_K3_KL_TR_ER &25
ORLD
ANDLD
OUT V0220_UT  ; Z
; rung 16: MOTTAK L2.2  V0247  TØM ETTER VASK
LD P_On
LDNOT HENGER02_DRIFT  ; XN4_BIL1_ i drift
AND L2_2_LINJETOEM_VASK  ; TOEM LINJE ETTER VASK
ANDNOT C10_IND_VST80_K3  ; Z
LD VST80_K3_0_STATUS  ; XX
AND C10_IND_VST80_K3  ; Z
AND=(300) _80_K3_KL_TR_ER &33
ORLD
ANDLD
OUT V0247_UT
; rung 17: SILO L1.1 - L1.2
; rung 18: SILO L2.1 - L2.2
; rung 19: Ingen_kommentar_funnet

### Section VENTILER_OPPSAMLING_UHT

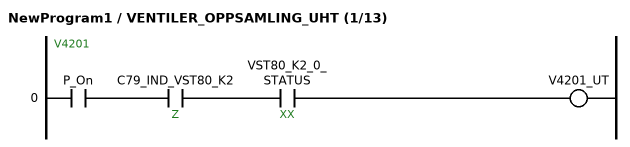
; rung 0: V4201
LD P_On
AND C79_IND_VST80_K2  ; Z
AND VST80_K2_0_STATUS  ; XX
OUT V4201_UT

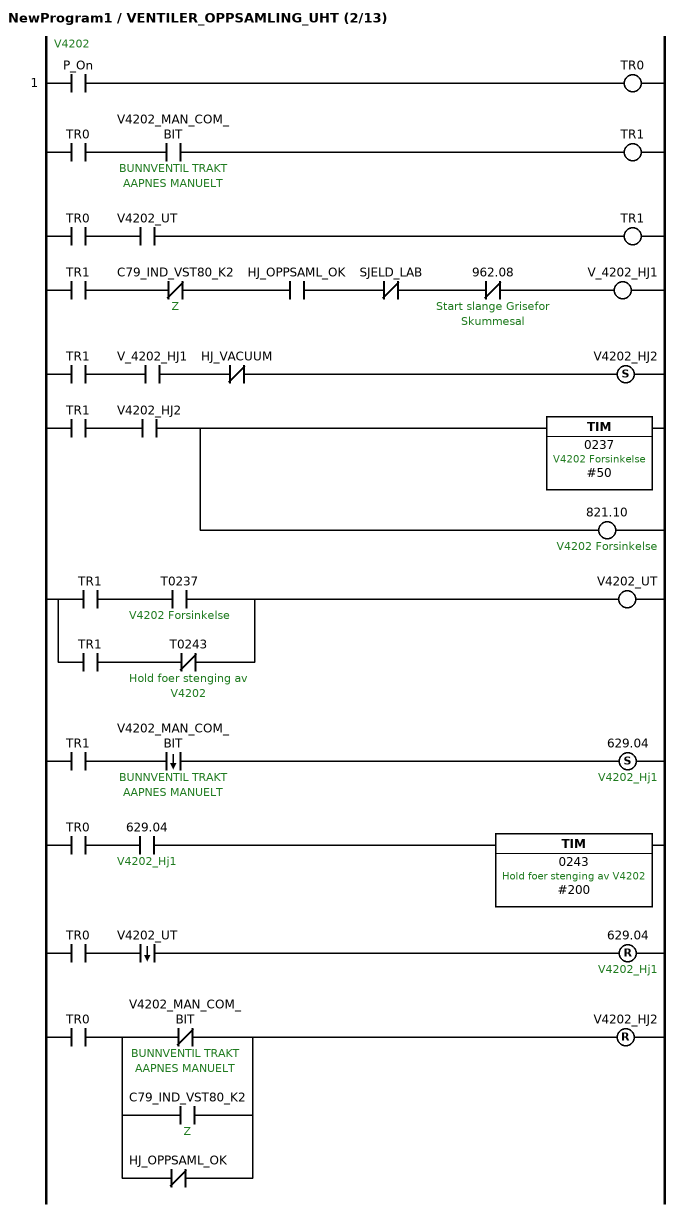
; rung 1: V4202
LD P_On
OUT TR0
AND V4202_MAN_COM_BIT  ; BUNNVENTIL TRAKT AAPNES MANUELT
OUT TR1
ANDNOT C79_IND_VST80_K2  ; Z
AND HJ_OPPSAML_OK
ANDNOT SJELD_LAB
ANDNOT 962.08  ; Start slange Grisefor Skummesal
OUT V_4202_HJ1
LD TR1
AND V_4202_HJ1
ANDNOT HJ_VACUUM
SET V4202_HJ2
LD TR1
AND V4202_HJ2
TIM 0237 #50  ; V4202 Forsinkelse
OUT 821.10  ; V4202 Forsinkelse
LD TR1
AND T0237  ; V4202 Forsinkelse
LD TR0
AND V4202_UT
OUT TR1
ANDNOT T0243  ; Hold foer stenging av V4202
ORLD
OUT V4202_UT
LD TR1
%AND V4202_MAN_COM_BIT  ; BUNNVENTIL TRAKT AAPNES MANUELT
SET 629.04  ; V4202_Hj1
LD TR0
AND 629.04  ; V4202_Hj1
TIM 0243 #200  ; Hold foer stenging av V4202
LD TR0
%AND V4202_UT
RSET 629.04  ; V4202_Hj1
LD TR0
LDNOT V4202_MAN_COM_BIT  ; BUNNVENTIL TRAKT AAPNES MANUELT
OR C79_IND_VST80_K2  ; Z
ORNOT HJ_OPPSAML_OK
ANDLD
RSET V4202_HJ2

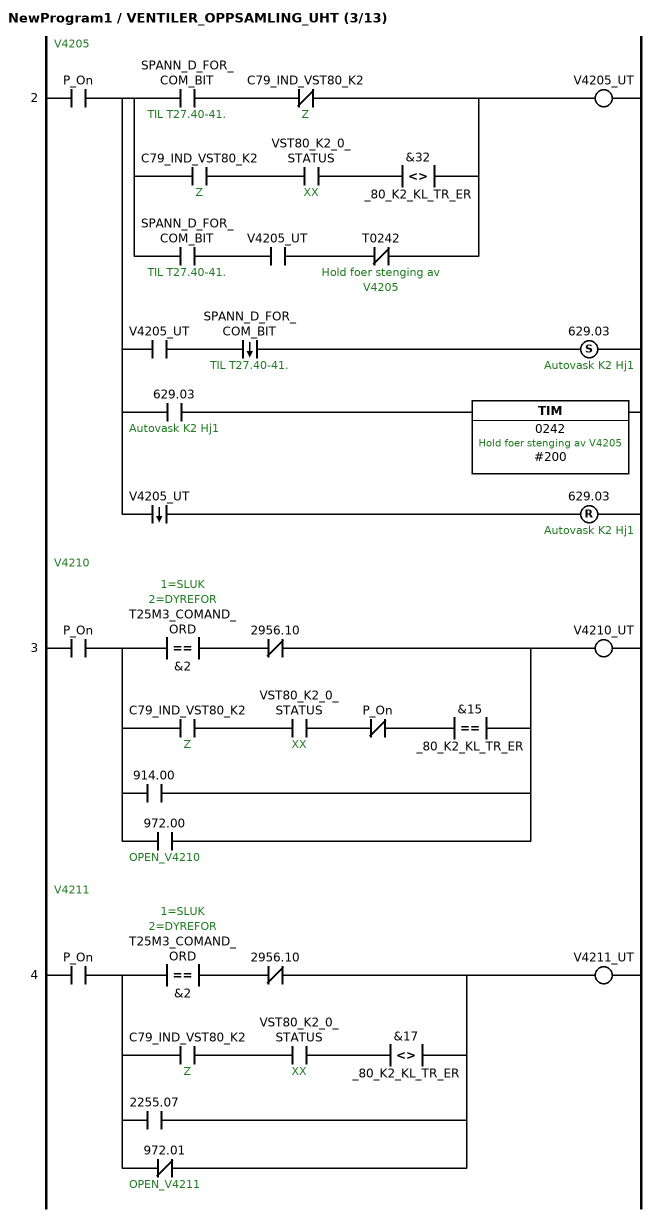
; rung 2: V4205
LD P_On
OUT TR0
LD SPANN_D_FOR_COM_BIT  ; TIL T27.40-41.
ANDNOT C79_IND_VST80_K2  ; Z
LD C79_IND_VST80_K2  ; Z
AND VST80_K2_0_STATUS  ; XX
AND<>(305) &32 _80_K2_KL_TR_ER
ORLD
LD SPANN_D_FOR_COM_BIT  ; TIL T27.40-41.
AND V4205_UT
ANDNOT T0242  ; Hold foer stenging av V4205
ORLD
ANDLD
OUT V4205_UT
LD TR0
AND V4205_UT
%AND SPANN_D_FOR_COM_BIT  ; TIL T27.40-41.
SET 629.03  ; Autovask K2 Hj1
LD TR0
AND 629.03  ; Autovask K2 Hj1
TIM 0242 #200  ; Hold foer stenging av V4205
LD TR0
%AND V4205_UT
RSET 629.03  ; Autovask K2 Hj1
; rung 3: V4210
LD P_On
LD=(300) T25M3_COMAND_ORD &2  ; 1=SLUK                                                                     2=DYREFOR
ANDNOT 2956.10
LD C79_IND_VST80_K2  ; Z
AND VST80_K2_0_STATUS  ; XX
ANDNOT P_On
AND=(300) &15 _80_K2_KL_TR_ER
ORLD
OR 914.00
OR 972.00  ; OPEN_V4210
ANDLD
OUT V4210_UT
; rung 4: V4211
LD P_On
LD=(300) T25M3_COMAND_ORD &2  ; 1=SLUK                                                                     2=DYREFOR
ANDNOT 2956.10
LD C79_IND_VST80_K2  ; Z
AND VST80_K2_0_STATUS  ; XX
AND<>(305) &17 _80_K2_KL_TR_ER
ORLD
OR 2255.07
ORNOT 972.01  ; OPEN_V4211
ANDLD
OUT V4211_UT

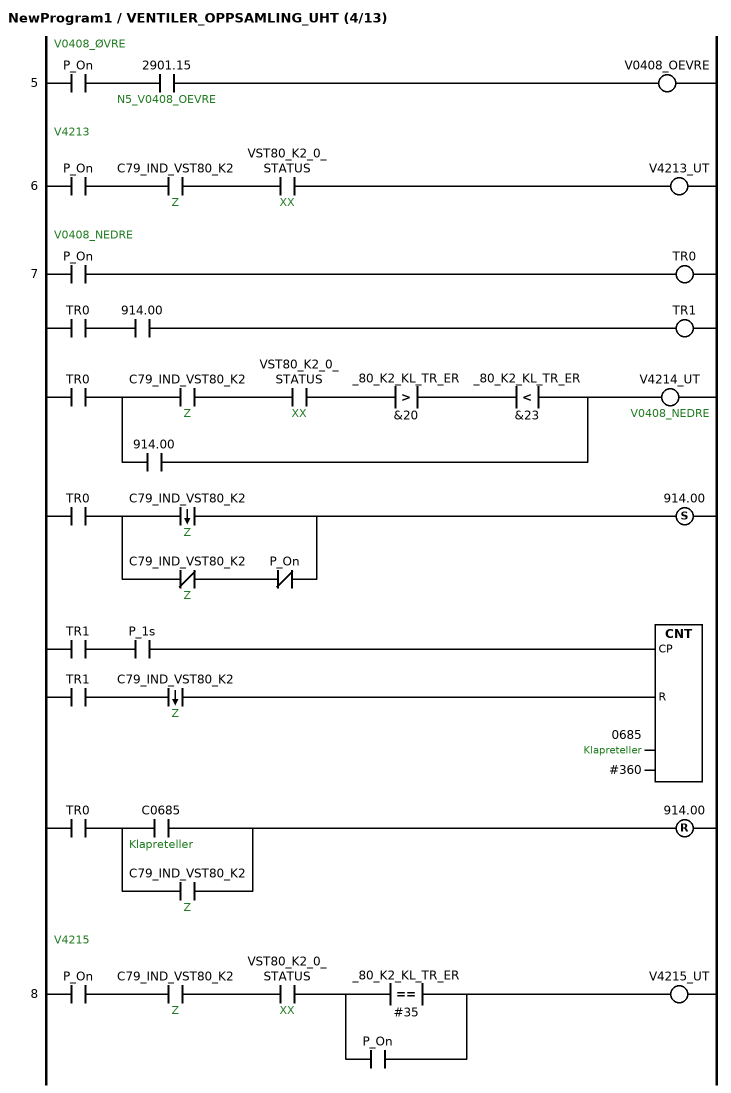
; rung 5: V0408_ØVRE
LD P_On
AND 2901.15  ; N5_V0408_OEVRE
OUT V0408_OEVRE
; rung 6: V4213
LD P_On
AND C79_IND_VST80_K2  ; Z
AND VST80_K2_0_STATUS  ; XX
OUT V4213_UT
; rung 7: V0408_NEDRE
LD P_On
OUT TR0
LD C79_IND_VST80_K2  ; Z
AND VST80_K2_0_STATUS  ; XX
AND>(320) _80_K2_KL_TR_ER &20
AND<(310) _80_K2_KL_TR_ER &23
OR 914.00
ANDLD
OUT V4214_UT  ; V0408_NEDRE
LD TR0
%LD C79_IND_VST80_K2  ; Z
LDNOT C79_IND_VST80_K2  ; Z
ANDNOT P_On
ORLD
ANDLD
SET 914.00
LD TR0
AND 914.00
OUT TR1
AND P_1s
LD TR1
%AND C79_IND_VST80_K2  ; Z
CNT 0685 #360  ; Klapreteller
LD TR0
LD C0685  ; Klapreteller
OR C79_IND_VST80_K2  ; Z
ANDLD
RSET 914.00
; rung 8: V4215
LD P_On
AND C79_IND_VST80_K2  ; Z
AND VST80_K2_0_STATUS  ; XX
LD=(300) _80_K2_KL_TR_ER #35
OR P_On
ANDLD
OUT V4215_UT

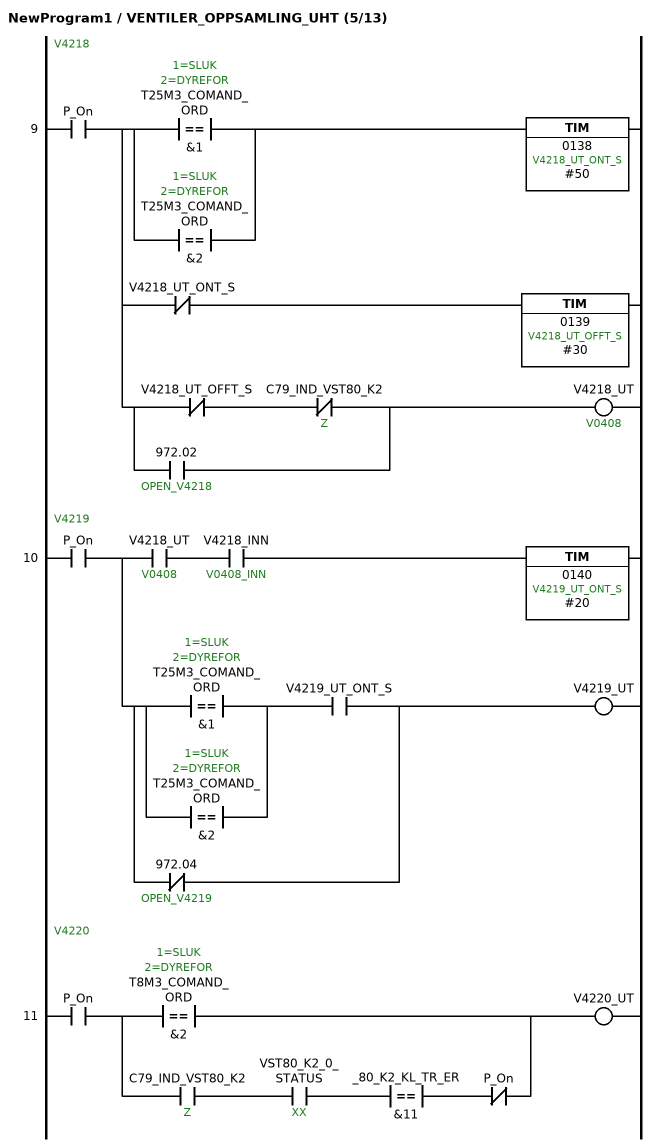
; rung 9: V4218
LD P_On
OUT TR0
LD=(300) T25M3_COMAND_ORD &1  ; 1=SLUK                                                                     2=DYREFOR
OR=(300) T25M3_COMAND_ORD &2  ; 1=SLUK                                                                     2=DYREFOR
ANDLD
TIM 0138 #50  ; V4218_UT_ONT_S
LD TR0
ANDNOT V4218_UT_ONT_S
TIM 0139 #30  ; V4218_UT_OFFT_S
LD TR0
LDNOT V4218_UT_OFFT_S
ANDNOT C79_IND_VST80_K2  ; Z
OR 972.02  ; OPEN_V4218
ANDLD
OUT V4218_UT  ; V0408
; rung 10: V4219
LD P_On
OUT TR0
AND V4218_UT  ; V0408
AND V4218_INN  ; V0408_INN
TIM 0140 #20  ; V4219_UT_ONT_S
LD TR0
LD=(300) T25M3_COMAND_ORD &1  ; 1=SLUK                                                                     2=DYREFOR
OR=(300) T25M3_COMAND_ORD &2  ; 1=SLUK                                                                     2=DYREFOR
AND V4219_UT_ONT_S
ORNOT 972.04  ; OPEN_V4219
ANDLD
OUT V4219_UT
; rung 11: V4220
LD P_On
LD=(300) T8M3_COMAND_ORD &2  ; 1=SLUK                                                                     2=DYREFOR
LD C79_IND_VST80_K2  ; Z
AND VST80_K2_0_STATUS  ; XX
AND=(300) _80_K2_KL_TR_ER &11
ANDNOT P_On
ORLD
ANDLD
OUT V4220_UT

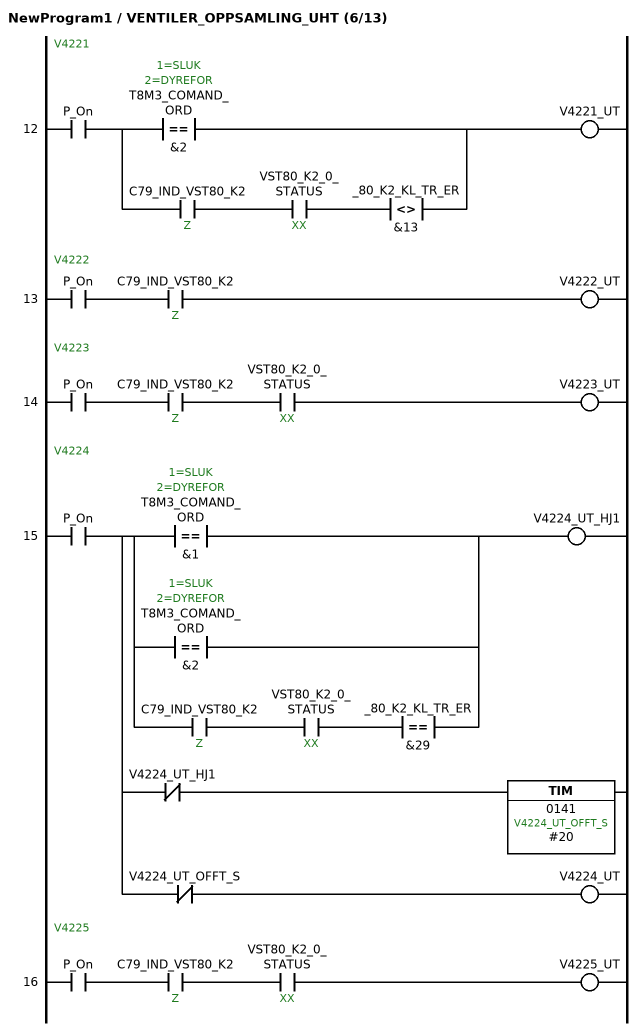
; rung 12: V4221
LD P_On
LD=(300) T8M3_COMAND_ORD &2  ; 1=SLUK                                                                     2=DYREFOR
LD C79_IND_VST80_K2  ; Z
AND VST80_K2_0_STATUS  ; XX
AND<>(305) _80_K2_KL_TR_ER &13
ORLD
ANDLD
OUT V4221_UT
; rung 13: V4222
LD P_On
AND C79_IND_VST80_K2  ; Z
OUT V4222_UT
; rung 14: V4223
LD P_On
AND C79_IND_VST80_K2  ; Z
AND VST80_K2_0_STATUS  ; XX
OUT V4223_UT
; rung 15: V4224
LD P_On
OUT TR0
LD=(300) T8M3_COMAND_ORD &1  ; 1=SLUK                                                                     2=DYREFOR
OR=(300) T8M3_COMAND_ORD &2  ; 1=SLUK                                                                     2=DYREFOR
LD C79_IND_VST80_K2  ; Z
AND VST80_K2_0_STATUS  ; XX
AND=(300) _80_K2_KL_TR_ER &29
ORLD
ANDLD
OUT V4224_UT_HJ1
LD TR0
ANDNOT V4224_UT_HJ1
TIM 0141 #20  ; V4224_UT_OFFT_S
LD TR0
ANDNOT V4224_UT_OFFT_S
OUT V4224_UT
; rung 16: V4225
LD P_On
AND C79_IND_VST80_K2  ; Z
AND VST80_K2_0_STATUS  ; XX
OUT V4225_UT

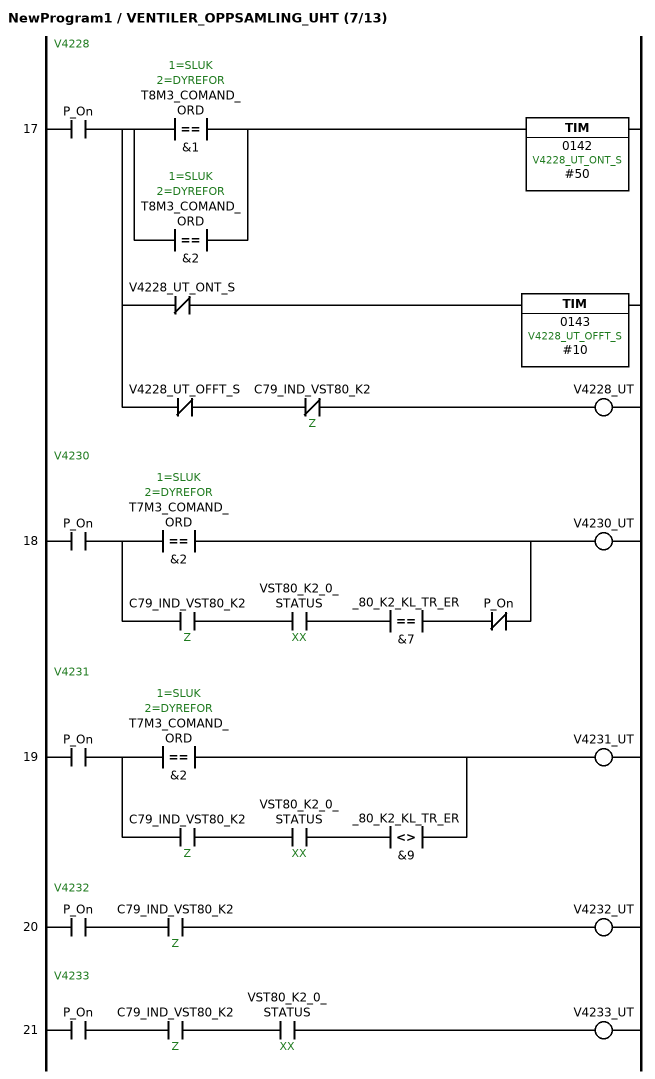
; rung 17: V4228
LD P_On
OUT TR0
LD=(300) T8M3_COMAND_ORD &1  ; 1=SLUK                                                                     2=DYREFOR
OR=(300) T8M3_COMAND_ORD &2  ; 1=SLUK                                                                     2=DYREFOR
ANDLD
TIM 0142 #50  ; V4228_UT_ONT_S
LD TR0
ANDNOT V4228_UT_ONT_S
TIM 0143 #10  ; V4228_UT_OFFT_S
LD TR0
ANDNOT V4228_UT_OFFT_S
ANDNOT C79_IND_VST80_K2  ; Z
OUT V4228_UT
; rung 18: V4230
LD P_On
LD=(300) T7M3_COMAND_ORD &2  ; 1=SLUK                                                                     2=DYREFOR
LD C79_IND_VST80_K2  ; Z
AND VST80_K2_0_STATUS  ; XX
AND=(300) _80_K2_KL_TR_ER &7
ANDNOT P_On
ORLD
ANDLD
OUT V4230_UT
; rung 19: V4231
LD P_On
LD=(300) T7M3_COMAND_ORD &2  ; 1=SLUK                                                                     2=DYREFOR
LD C79_IND_VST80_K2  ; Z
AND VST80_K2_0_STATUS  ; XX
AND<>(305) _80_K2_KL_TR_ER &9
ORLD
ANDLD
OUT V4231_UT
; rung 20: V4232
LD P_On
AND C79_IND_VST80_K2  ; Z
OUT V4232_UT
; rung 21: V4233
LD P_On
AND C79_IND_VST80_K2  ; Z
AND VST80_K2_0_STATUS  ; XX
OUT V4233_UT

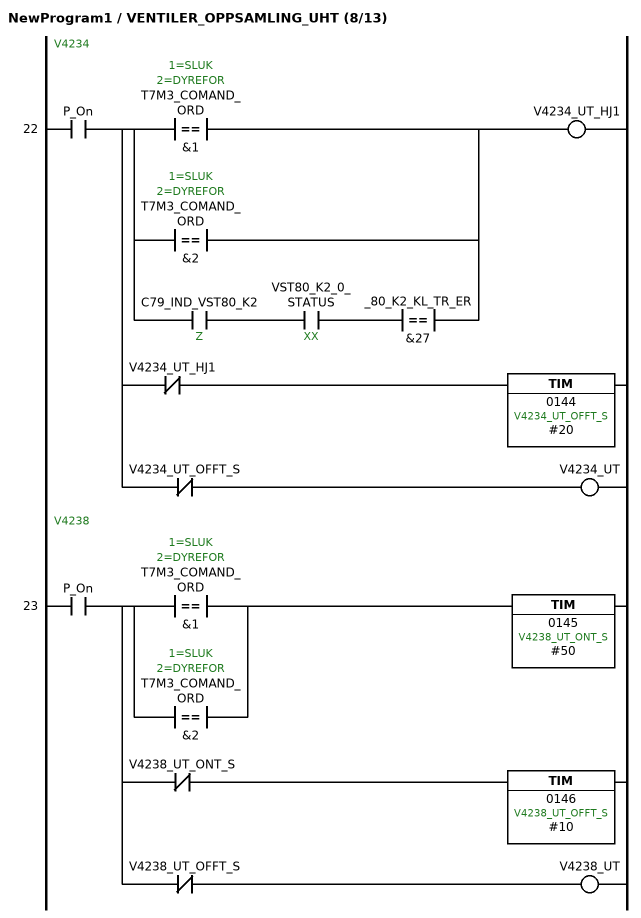
; rung 22: V4234
LD P_On
OUT TR0
LD=(300) T7M3_COMAND_ORD &1  ; 1=SLUK                                                                     2=DYREFOR
OR=(300) T7M3_COMAND_ORD &2  ; 1=SLUK                                                                     2=DYREFOR
LD C79_IND_VST80_K2  ; Z
AND VST80_K2_0_STATUS  ; XX
AND=(300) _80_K2_KL_TR_ER &27
ORLD
ANDLD
OUT V4234_UT_HJ1
LD TR0
ANDNOT V4234_UT_HJ1
TIM 0144 #20  ; V4234_UT_OFFT_S
LD TR0
ANDNOT V4234_UT_OFFT_S
OUT V4234_UT
; rung 23: V4238
LD P_On
OUT TR0
LD=(300) T7M3_COMAND_ORD &1  ; 1=SLUK                                                                     2=DYREFOR
OR=(300) T7M3_COMAND_ORD &2  ; 1=SLUK                                                                     2=DYREFOR
ANDLD
TIM 0145 #50  ; V4238_UT_ONT_S
LD TR0
ANDNOT V4238_UT_ONT_S
TIM 0146 #10  ; V4238_UT_OFFT_S
LD TR0
ANDNOT V4238_UT_OFFT_S
OUT V4238_UT

